(* Logix 5000 project; controller miPrimerPrograma Emulate 5570 rev 32.11; software revision 32.02 *)

TASK T00_MainTask (continuous, watchdog 500 ms) : P00_MainProgram

MODULES
   Local : Emulate 5570 (ICP 2, rev 32.11)
END_MODULES

VAR_GLOBAL   (* controller tags *)
   botonArranque : BOOL;
   botonParo : BOOL := 1;
   entrada1 : BOOL := 1;   // memoriaVirtual
   entrada2 : BOOL := 1;   // memoriaVirtual
   motor : BOOL;
   salida1 : BOOL := 1;   // memoriaVirual
END_VAR

PROGRAM P00_MainProgram   (* main routine R00_MainRoutine *)
VAR
   salida2 : BOOL := 1;
END_VAR

ROUTINE R00_MainRoutine   (* ladder *)
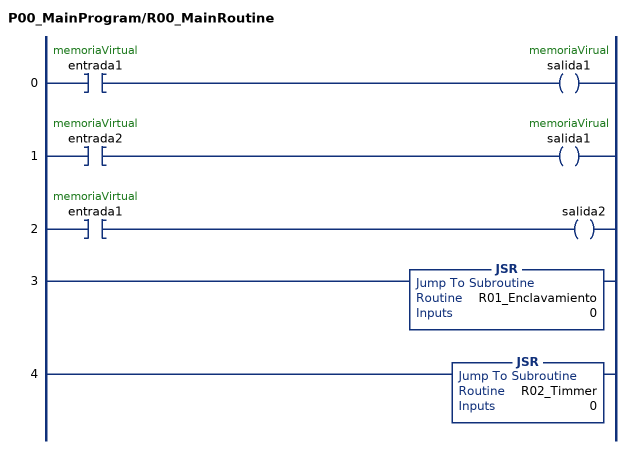
   0: XIC(entrada1)OTE(salida1);
   1: XIC(entrada2)OTE(salida1);
   2: XIC(entrada1)OTE(salida2);
   3: JSR(R01_Enclavamiento,0);
   4: JSR(R02_Timmer,0);
END_ROUTINE

ROUTINE R01_Enclavamiento   (* ladder *)
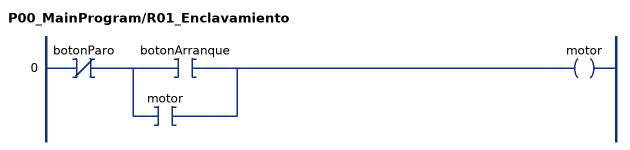
   0: XIO(botonParo)[XIC(botonArranque) ,XIC(motor) ]OTE(motor);
END_ROUTINE

ROUTINE R02_Timmer   (* ladder *)
   0: ;
END_ROUTINE
END_PROGRAM
